Fanuc KAREL source: webabort.kl

PROGRAM webabort
%COMMENT = 'v3'
%NOLOCKGROUP
%NOPAUSE=ERROR+COMMAND+TPENABLE
%NOBUSYLAMP

CONST

	PR_WEBJOINTS = 40
	PR_WEBXYZWPR = 41

	R_WEBKEEP = 42

VAR

	STATUS: INTEGER
	return_code: INTEGER

	cur_jpos: JOINTPOS
	cur_pos: XYZWPR

BEGIN

	WRITE (CHR(128),CHR(137))

	ABORT_TASK('*ALL*', TRUE, TRUE, STATUS)

	IF (STATUS <> 0 ) THEN
		WRITE ('ABORT_TASK built-IN failed WITH STATUS = ', STATUS, CR)
	ENDIF

	cur_jpos = CURJPOS(0,0)
	cur_pos = CURPOS(0,0)

	SET_JPOS_REG(PR_WEBJOINTS, cur_jpos, STATUS)

	IF (STATUS <> 0 ) THEN
		WRITE ('SET_JPOS_REG built-IN failed in ABORT task WITH STATUS = ', STATUS, CR)
	ENDIF

	SET_POS_REG(PR_WEBXYZWPR, cur_pos, STATUS)

	IF (STATUS <> 0 ) THEN
		WRITE ('SET_POS_REG built-IN failed in ABORT task WITH STATUS = ', STATUS, CR)
	ENDIF

	FLG[1] = OFF
	FLG[2] = OFF
	FLG[3] = OFF
	FLG[4] = OFF
	FLG[5] = OFF
	FLG[6] = OFF
	FLG[7] = OFF
	FLG[8] = OFF

	SET_REAL_REG(R_WEBKEEP, 999, STATUS)

	IF (STATUS <> 0 ) THEN
		WRITE ('SET_REL_REG built-IN 3 failed: ', STATUS, CR)
	ENDIF

	CLEAR('webmonitor.pc', STATUS)

	IF (STATUS <> 0 ) THEN
		WRITE ('CLEAR  built-IN failed: ', STATUS, CR)
	ENDIF

	return_code = 204

END webabort
